// TIA Portal V19 export
DATA_BLOCK "Production"   // DB7
// stored: MemoryReserve 100
   VAR RETAIN
      Last_O_ID { ExternalWritable := 'False'} : DInt;   // Ultmo ID assegnato a un ProdItem
      O_Empty { ExternalWritable := 'False'} : "Prod_Item";   // Ordine vuoto per operrazioni di cancellazione
      O_ACT { ExternalWritable := 'False'} : "Prod_Item";   // ORDINE CON PARTI IN ESECUZIONE AL TAGLIO
      O_TODO { ExternalWritable := 'False'} : Array[1.."PROD_TODO_ITEMS"] of "Prod_Item";   // LISTA CON ORDINI DI PRODUZIONE PRONTI PER ESSERE ESEGUI
      O_ENDING { ExternalWritable := 'False'} : Array[1.."PROD_ENDING_ITEMS"] of "Prod_Item";   // ORDINI NON PIU' AL TAGLIO & NON USCITI DAL PROCESSO
      O_OUT { ExternalWritable := 'False'} : Array[1.."PROD_OUT_ITEMS"] of "Prod_Item";   // ORDINI / PEZZI USCITI DAL PROCESSO
      Coil_Data { ExternalWritable := 'False'} : Struct
         Last_C_ID : DInt;
         Empty : "Coil_Item";
         ASPO_IN_CARICO : "Coil_Item";
         ASPO_IN_LINEA : "Coil_Item";
         JB : "Coil_Item";
         TAGLIO_FINALE : "Coil_Item";
         OUT { S7_SetPoint := 'True'} : Array[1.."PROD_COILS_OUT_ITEMS"] of "Coil_Item";
      END_STRUCT;
   END_VAR
BEGIN
END_DATA_BLOCK
